FUNCTION_BLOCK TankCtrl IMPLEMENTS I_Domain, I_Execute
VAR_INPUT
	bNoWater		: BOOL;
	bOverload		: BOOL;
END_VAR
VAR_OUTPUT
	bRunPump		: BOOL;
END_VAR
VAR CONSTANT
	MAX_STATE		: UDINT := 5;
END_VAR
VAR
	exe				: Execute(THIS^);

	// Context
	ctx				: TankCtrl_Ctx;

	// State Machine
	
	stateMachine	: StateMachine;
	stateRepo		: StateRepo<MAX_STATE>;
	stateBuffer		: StateBuffer<MAX_STATE>;
	stateMgr		: StateManager<MAX_STATE>(stateMachine, stateRepo, stateBuffer);
	A_Smgr			: A_StateManager(stateMgr, ctx.priv.smgr);
	
	// States	
	EStop			: TankCtrl_EStop(stateRepo, ctx);
	A_EStop			: A_Tag(EStop.Tag, ctx.state.iEStop);
	OnEStop			: Receiver(EStop);
	
	Disabled		: TankCtrl_Disabled(stateRepo, ctx);
	A_Disabled		: A_Tag(Disabled.Tag, ctx.state.iDisabled);
	
	Fault			: TankCtrl_Fault(stateRepo, ctx);
	A_Fault			: A_Tag(Fault.Tag, ctx.state.iFault);
	
	Enabled			: TankCtrl_Enabled(stateRepo, ctx);
	A_Enabled		: A_Tag(Enabled.Tag, ctx.state.iEnabled);
	OnRequest		: Receiver(Enabled);

	Filling			: TankCtrl_Filling(stateRepo, ctx);
	A_Filling		: A_Tag(Filling.Tag, ctx.state.iFilling);
	
	// FLAGS
	flagList		: FlagList<1>;
	A_SystemOn		: A_Flag(flagList, ctx.priv.IsSystemOn);
	
	// SIGNALS
	signalList		: SignalList<1>;
	A_SmgrChange	: A_Signal(signalList, stateMgr.GetOnChange());
	
	// RECEIVERS
	receiverList	: ReceiverList<2>;
	A_OnEStop		: A_Receiver(receiverList, OnEStop);
	A_OnRequest		: A_Receiver(receiverList, OnRequest);
	
	// HMI
	statusText		: TankCtrl_StatusText(ctx);
	
	// DOMAIN
	domTag			: Tag;
	domain			: Domain(domTag, stateMgr, flagList, signalList, receiverList);
	
	// PRIV
	bInit			: BOOL := TRUE;
END_VAR

METHOD Execute
IF bInit THEN
	ctx.priv.smgr.Request(ctx.state.iDisabled);	

	bInit := FALSE;
END_IF

// INPUTS
ctx.io.in.bNoWater := bNoWater;
ctx.io.in.bOverload := bOverload;

// OUTPUTS
bRunPump := ctx.io.out.bRunPump;
END_METHOD

PROPERTY Flags : Domains.Flags.I_FlagList
GET
Flags := flagList;
END_GET
END_PROPERTY

PROPERTY Recs : Domains.Broadcast.I_ReceiverList
GET
Recs := receiverList;
END_GET
END_PROPERTY

PROPERTY Signals : Domains.Broadcast.I_SignalList
GET
Signals := signalList;
END_GET
END_PROPERTY

PROPERTY Smgr : Domains.States.I_StateManager
GET
Smgr := stateMgr;
END_GET
END_PROPERTY

PROPERTY Tag : Tags.I_Tag
GET
Tag := domTag;
END_GET
END_PROPERTY

METHOD ToDebug : Debug.I_Debug
ToDebug := THIS^;
END_METHOD

END_FUNCTION_BLOCK

(* stored: Version 1.1.0.1
   POU TankCtrl: Id {71dfe158-063e-4ac3-bf98-44fac6c2f0af}, SpecialFunc None
   Method Execute: Id {93d893b4-6efe-4ab4-94a5-1399cd89b222}
   Property Flags: Id {daf66693-a007-483b-8839-5471e7be9f40}
   Get Get: Id {0b3b47b4-7123-4393-b2fe-8438ae01be66}
   Property Recs: Id {6b826d4b-2a86-4d78-8b9b-deed25c411b1}
   Get Get: Id {2fd752c6-4e7a-4f6e-8be5-6abdf451a764}
   Property Signals: Id {d105e1ef-7f07-4886-acbf-6c59b5817d87}
   Get Get: Id {0098bed3-4745-4ac4-a82f-6a07b4649e23}
   Property Smgr: Id {7c9ac3ef-c213-4a70-b242-4aa5a787835c}
   Get Get: Id {7639a792-8ea8-4c60-ac61-9773a983d77d}
   Property Tag: Id {515a06bf-72bb-407b-a993-161476064e14}
   Get Get: Id {ba92eba2-b38b-4db5-8536-c654f0547753}
   Method ToDebug: Id {23787608-9066-4bff-8e91-0fe971cc4889} *)
